Universal Robots PolyScope program: get_pose.urp

Program get_pose (installation=default directory=/programs createdIn=5.2.0.61336 lastSavedIn=5.2.0.61336 robotSerialNumber=20185300040)
Calibrated DH parameters: a=[-0.000128, -0.221415, -0.194849, 0.000098, -0.000148, 0]; d=[0.152137, 33.879231, 13.968137, -47.716378, 0.085395, 0.092257]; alpha=[1.57105, 0.003021, -0.001826, 1.571145, -1.57192, 0]; deltaTheta=[0, 0.433042, -0.854582, 0.421536, 0.000002, 0]
Robot Program (runOnlyOnce=false)
  var_1 := get_actual_tcp_pose()
  Wait Sleep waitTime=0.01
